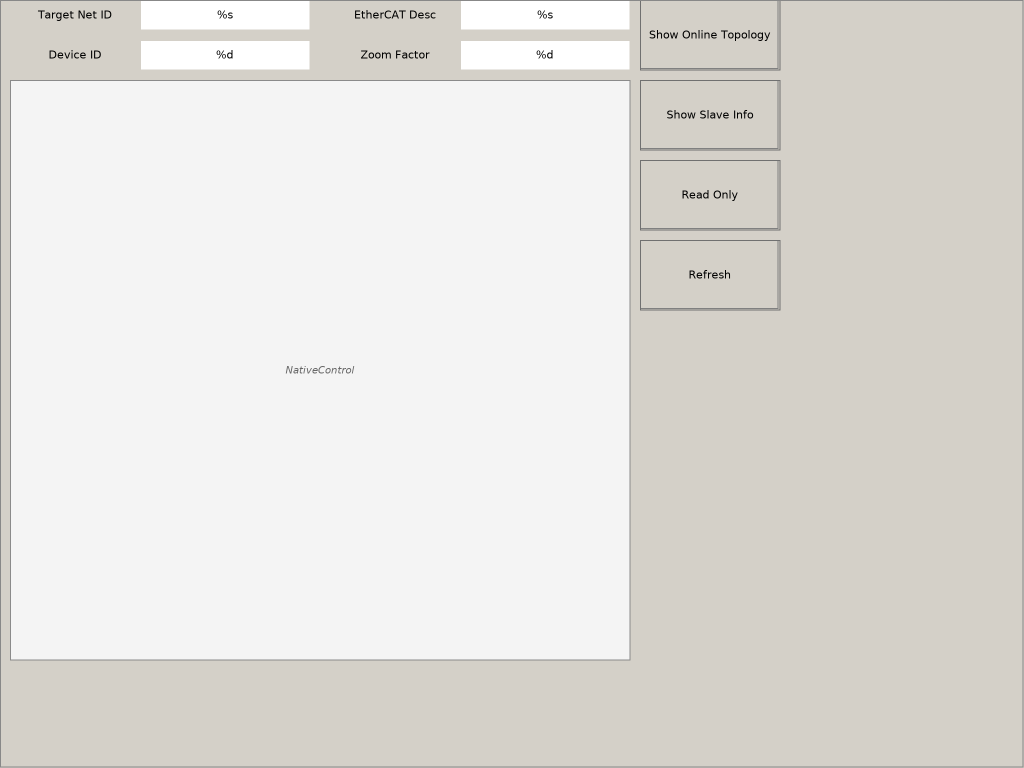
VISUALIZATION Visualization  // 1024x768
    NativeControl (10,80 620x580)
        Calls[0]: Method=TargetNetId, Method=ShowOnlineTopology, Variable=MAIN.bShowOnlineTopology
        Parameters[0]: Var=MAIN.sTargetNetID, Var=MAIN.udiDeviceID, Var=MAIN.udiZoomFactor, Var=MAIN.bSowSlaveInfo, Var=MAIN.sSlaveDescriptionPath, Var=MAIN.bReadOnly
        Calls[1]: Method=DeviceId, Method=ZoomFactor, Variable=MAIN.bRefresh
        Calls[2]: Method=SlaveDescriptionPath, Method=ShowSlaveInfo, Variable=MAIN.bSowSlaveInfo
        Calls[3]: Method=ReadOnly, Variable=MAIN.bRefresh
        p3873840581: EcTopology.EcTopologyCtrl.1
    Button (640,0 140x70), "Show Online Topology"
        tap MAIN.bShowOnlineTopology
    Textfield (140,0 170x30), "%s", text variable: MAIN.sTargetNetID
        OnMouseClick: write the text variable via Default
    Label (0,0 150x30), "Target Net ID"
    Textfield (140,40 170x30), "%d", text variable: MAIN.udiDeviceID
        OnMouseClick: write the text variable via Default
    Label (0,40 150x30), "Device ID"
    Textfield (460,0 170x30), "%s", text variable: MAIN.sSlaveDescriptionPath
        OnMouseClick: write the text variable via Default
    Label (320,0 150x30), "EtherCAT Desc"
    Textfield (460,40 170x30), "%d", text variable: MAIN.udiZoomFactor
        OnMouseClick: write the text variable via Default
    Label (320,40 150x30), "Zoom Factor"
    Button (640,80 140x70), "Show Slave Info"
        toggle MAIN.bSowSlaveInfo
    Button (640,160 140x70), "Read Only"
        tap MAIN.bRefresh
    Button (640,240 140x70), "Refresh"
        tap MAIN.bRefresh
END_VISUALIZATION

(* stored: Version 1.1.0.1, ProductVersion 3.1.4024.3
   Visu Visualization: Id {2926713d-cb96-480c-8e94-62e95ff9c353} *)
